(* CODESYS project Files.library
   Title: Files
   Version: 0.0.1
   Placeholder: Files
   Company: TomasRompotl

Project tree, tasks and I/O mapping:
  libraries: Events, * (TomasRompotl); MachineBase, * (TomasRompotl); Tc2_Standard, * (Beckhoff Automation GmbH); Tc2_System, * (Beckhoff Automation GmbH); Tc2_Utilities, * (Beckhoff Automation GmbH); Tc3_Module, * (Beckhoff Automation GmbH)
  File/
    function block Directory [ST]: Abort, Create, Cyclic, FileExists, FileNameList, CheckFileExists, List, Remove
    function block File [ST]: Busy, Cyclic, Done, Error, Read, Write
    function block FileRemover [ST]: Busy, Cyclic, Done, Error, Remove
  Version/
    global variables Global_Version
*)

// Version/Global_Version
{attribute 'TcGenerated'}
{attribute 'no-analysis'}
{attribute 'linkalways'}
// This function has been automatically generated from the project information.
VAR_GLOBAL CONSTANT
	{attribute 'const_non_replaced'}
	stLibVersion_Files : ST_LibVersion := (iMajor := 0, iMinor := 0, iBuild := 1, iRevision := 0, nFlags := 0, sVersion := '0.0.1');
END_VAR

// File/Directory
FUNCTION_BLOCK Directory
VAR
	creator : FB_CreateDir; // can only create on level of folder
	remover : FB_RemoveDir; // can only remove topmost folder. Not folder with folders.

	listDir : FB_EnumFindFileList;	
	listingFinishedTrigger : F_TRIG;
	fileListDone : BOOL;
	checkingFolder : BOOL;
	checkingFileExistence : BOOL;

	page : ARRAY[0..50 - 1] OF ST_FindFileEntry;
	_FileNameList : ARRAY[0..50 - 1] OF T_MaxString;
	_FileExists : BOOL;
	
	createDirectoryErrorTrig : R_TRIG;
	removeDirectoryErrorTrig : R_TRIG;
	listingDirectoryErrorTrig : R_TRIG;
	createDirectoryError : MessageEventLogger(TC_EVENTS.DirectoryEventClass.CreateDirectoryError);
	removeDirectoryError : MessageEventLogger(TC_EVENTS.DirectoryEventClass.RemoveDirectoryError);
	listingDirectoryError : MessageEventLogger(TC_EVENTS.DirectoryEventClass.ListDirectoryError);
END_VAR
VAR CONSTANT
	EntriesPerPage : INT := 50;
END_VAR

METHOD PRIVATE Abort
VAR_INPUT
END_VAR
listDir(
	bExecute := TRUE,
	eCmd := E_EnumCmdType.eEnumCmd_Abort
);
listDir(bExecute := FALSE);
END_METHOD

{attribute 'TcRpcEnable':='1'}
METHOD Create
VAR_INPUT
	path : T_MaxString;
END_VAR
creator(
	sPathName := path,
	bExecute := TRUE,
);
END_METHOD

METHOD Cyclic
VAR
	i : INT;
END_VAR
creator(bExecute := FALSE);
remover(bExecute := FALSE);

listDir(
	pFindList := ADR(page),
	cbFindList := SIZEOF(page)
);

listingFinishedTrigger(CLK := listDir.bBusy);
IF (listingFinishedTrigger.Q AND listDir.eCmd <> E_EnumCmdType.eEnumCmd_Abort) THEN

	listDir(bExecute := FALSE);
	fileListDone := TRUE;
	
	FOR i := 0 TO EntriesPerPage - 1 DO
		_FileNameList[i] := page[i].sFileName;
		
		IF (checkingFileExistence) THEN
			IF (page[i].fileAttributes.bDirectory = checkingFolder
				AND page[i].sFileName <> '') THEN
				_FileExists := TRUE;
			END_IF
		END_IF
	END_FOR
	
	IF (NOT listDir.bEOE) THEN
		Abort();
	END_IF
END_IF

createDirectoryErrorTrig(CLK := creator.bError);
removeDirectoryErrorTrig(CLK := remover.bError);
listingDirectoryErrorTrig(CLK := listDir.bError);
IF (createDirectoryErrorTrig.Q) THEN
	createDirectoryError.Arguments.Clear().AddStringByValue(creator.sPathName);
	createDirectoryError.Send();
END_IF
IF (removeDirectoryErrorTrig.Q) THEN
	removeDirectoryError.Arguments.Clear().AddStringByValue(remover.sPathName);
	removeDirectoryError.Send();
END_IF
IF (listingDirectoryErrorTrig.Q) THEN
	listingDirectoryError.Arguments.Clear().AddStringByValue(listDir.sPathName);
	listingDirectoryError.Send();
END_IF
END_METHOD

{attribute 'monitoring' := 'call'}
PROPERTY FileExists : BOOL
GET
FileExists := _FileExists;
END_GET
END_PROPERTY

{attribute 'monitoring' := 'call'}
PROPERTY FileNameList : REFERENCE TO ARRAY[0..49] OF T_MaxString
GET
FileNameList REF= _FileNameList;
END_GET
END_PROPERTY

METHOD CheckFileExists
VAR_INPUT
	path : T_MaxString;
	folder : BOOL; // FALSE = File, TRUE = Folder
END_VAR
IF (NOT listDir.bBusy) THEN
	
	List(path);
	
	_FileExists := FALSE;
	checkingFileExistence := TRUE;
	checkingFolder := folder;
END_IF
END_METHOD

 // Usage of * wildcard recommended
 // Add * to the end of path to list all files
METHOD List
VAR_INPUT
	path : T_MaxString;
END_VAR
IF (NOT listDir.bBusy) THEN
	
	checkingFileExistence := FALSE;
	fileListDone := FALSE;
	
	listDir(bExecute := FALSE);
	listDir(
		sPathName := path,
		eCmd := E_EnumCmdType.eEnumCmd_First,
		bExecute := TRUE
	);
END_IF
END_METHOD

METHOD Remove
VAR_INPUT
	path : T_MaxString;
END_VAR
remover(
	sPathName := path,
	bExecute := TRUE,
);
END_METHOD

END_FUNCTION_BLOCK

// File/File
FUNCTION_BLOCK File IMPLEMENTS Cyclic
VAR
	_Busy : BOOL;
	_Done : BOOL;
	_Error : BOOL;
	
	openRequest : BOOL;
	readRequest : BOOL;
	writeRequest : BOOL;
	appendMode : BOOL;
	filePath : T_MaxString;
	
	buffer : POINTER TO BYTE;
	bufferLength : UDINT;

	handle : UINT;
	opener : FB_FileOpen;
	closer : FB_FileClose;
	reader : FB_FileRead;
	writer : FB_FileWrite;
	
	fileState : (Waiting, OpenMode, Opening, Reading, Writing, Closing);
	openErrorTrigger : R_TRIG;
	readErrorTrigger : R_TRIG;
	writeErrorTrigger : R_TRIG;
	closeErrorTrigger : R_TRIG;
	
	notFoundError : MessageEventLogger(TC_EVENTS.FileEventClass.InvalidPath);
	fileOpenError : MessageEventLogger(TC_EVENTS.FileEventClass.OpenFileError);
	fileReadError : MessageEventLogger(TC_EVENTS.FileEventClass.ReadFileError);
	fileWriteError : MessageEventLogger(TC_EVENTS.FileEventClass.WriteFileError);
	fileCloseError : MessageEventLogger(TC_EVENTS.FileEventClass.CloseFileError);
END_VAR
VAR CONSTANT
	NotFoundErrorNumber : UDINT := 16#70C;
END_VAR

{attribute 'monitoring' := 'call'}
PROPERTY Busy : BOOL
GET
Busy := _Busy;
END_GET
END_PROPERTY

METHOD Cyclic
CASE fileState OF
	
	Waiting:
	
		IF (openRequest) THEN
			openRequest := FALSE;
			_Done := FALSE;
			
			fileState := OpenMode;
		END_IF
	
	OpenMode:
	
		IF (readRequest) THEN
			opener.nMode := FOPEN_MODEREAD;
		ELSIF (writeRequest) THEN
			IF (appendMode) THEN
				opener.nMode := FOPEN_MODEAPPEND;
			ELSE
				opener.nMode := FOPEN_MODEWRITE;
			END_IF
		END_IF
		
		opener.nMode := opener.nMode OR FOPEN_MODETEXT;

		fileState := Opening;
	
	Opening:
	
		opener(
			bExecute := NOT opener.bBusy,
			sPathName := filePath,
			hFile => handle,
		);
		
		IF (NOT opener.bExecute AND NOT opener.bBusy AND handle <> 0) THEN
			opener();
			IF (readRequest) THEN
				fileState := Reading;
			ELSIF (writeRequest) THEN
				fileState := Writing;
			END_IF
		END_IF
	
	Reading:
	
		reader(
			bExecute := NOT reader.bBusy,
			hFile := handle,
			pReadBuff := buffer,
			cbReadLen := bufferLength,
		);
		
		IF (NOT reader.bExecute AND NOT reader.bBusy) THEN
			fileState := Closing;
		END_IF
	
	Writing:
	
		writer(
			bExecute := NOT writer.bBusy,
			hFile := handle,
			pWriteBuff := buffer,
			cbWriteLen := bufferLength,
		);
		
		IF (NOT writer.bExecute AND NOT writer.bBusy) THEN
			fileState := Closing;
		END_IF
	
	Closing:
	
		IF (handle = 0) THEN
			fileState := Waiting;
		ELSE
			closer(
				bExecute := NOT closer.bBusy,
				hFile := handle,
			);
			
			IF (NOT closer.bExecute AND NOT closer.bBusy) THEN
				closer();
				handle := 0;
				_Done := TRUE;
				
				fileState := Waiting;
			END_IF
		END_IF
	
END_CASE

_Busy := fileState <> Waiting;

openErrorTrigger(CLK := opener.bError);
readErrorTrigger(CLK := reader.bError);
writeErrorTrigger(CLK := writer.bError);
closeErrorTrigger(CLK := closer.bError);
_Error := 
	openErrorTrigger.Q
	OR readErrorTrigger.Q
	OR writeErrorTrigger.Q
	OR closeErrorTrigger.Q
	;
IF (_Error) THEN
	openRequest := FALSE;
	readRequest := FALSE;
	writeRequest := FALSE;
	
	IF (openErrorTrigger.Q AND opener.nErrId = NotFoundErrorNumber) THEN
		notFoundError.Arguments.Clear().AddStringByValue(opener.sPathName);
		notFoundError.Send();
	ELSIF (openErrorTrigger.Q) THEN
		fileOpenError.Arguments.Clear().AddStringByValue(opener.sPathName);
		fileOpenError.Send();
	ELSIF (readErrorTrigger.Q) THEN
		fileReadError.Arguments.Clear().AddStringByValue(opener.sPathName);
		fileReadError.Send();
	ELSIF (openErrorTrigger.Q) THEN
		fileWriteError.Arguments.Clear().AddStringByValue(opener.sPathName);
		fileWriteError.Send();
	ELSIF (openErrorTrigger.Q) THEN
		fileCloseError.Arguments.Clear().AddStringByValue(opener.sPathName);
		fileCloseError.Send();
	END_IF
	
	IF (fileState > Waiting AND fileState < Closing) THEN
		fileState := Closing;
	END_IF
END_IF
END_METHOD

{attribute 'monitoring' := 'call'}
PROPERTY Done : BOOL
GET
Done := _Done;
END_GET
END_PROPERTY

{attribute 'monitoring' := 'call'}
PROPERTY Error : BOOL
GET
Error := _Error;
END_GET
END_PROPERTY

METHOD Read
VAR_INPUT
	buffer : POINTER TO BYTE;
	bufferLength : UDINT;
	filePath : T_MaxString;
END_VAR
IF (NOT _Busy) THEN
	THIS^.filePath := filePath;
	THIS^.buffer := buffer;
	THIS^.bufferLength := bufferLength;
	
	openRequest := TRUE;
	readRequest := TRUE;
	writeRequest := FALSE;
END_IF
END_METHOD

METHOD Write
VAR_INPUT
	buffer : POINTER TO BYTE;
	bufferLength : UDINT;
	filePath : T_MaxString;
	append : BOOL;
END_VAR
IF (NOT _Busy) THEN
	THIS^.filePath := filePath;
	THIS^.buffer := buffer;
	THIS^.bufferLength := bufferLength;
	
	openRequest := TRUE;
	writeRequest := TRUE;
	readRequest := FALSE;
	appendMode := append;
END_IF
END_METHOD

END_FUNCTION_BLOCK

// File/FileRemover
FUNCTION_BLOCK FileRemover IMPLEMENTS Cyclic
VAR
	remover : FB_FileDelete;
	
	removeErrorTrigger : R_TRIG;
	notFoundError : MessageEventLogger(TC_EVENTS.FileEventClass.InvalidPath);
	removeError : MessageEventLogger(TC_EVENTS.FileEventClass.RemoveFileError);
END_VAR
VAR CONSTANT
	NotFoundErrorNumber : UDINT := 16#70C;
END_VAR

{attribute 'monitoring' := 'call'}
PROPERTY Busy : BOOL
GET
Busy := remover.bBusy;
END_GET
END_PROPERTY

METHOD Cyclic
remover(bExecute := FALSE);

removeErrorTrigger(CLK := remover.bError);
IF (removeErrorTrigger.Q) THEN
	IF (remover.nErrId = NotFoundErrorNumber) THEN
		notFoundError.Arguments.Clear().AddStringByValue(remover.sPathName);
		notFoundError.Send();
	ELSE
		removeError.Arguments.Clear().AddStringByValue(remover.sPathName);
		removeError.Send();
	END_IF
END_IF
END_METHOD

{attribute 'monitoring' := 'call'}
PROPERTY Done : BOOL
GET
Done := NOT remover.bBusy;
END_GET
END_PROPERTY

{attribute 'monitoring' := 'call'}
PROPERTY Error : BOOL
GET
Error := remover.bError;
END_GET
END_PROPERTY

METHOD Remove
VAR_INPUT
	filePath : T_MaxString;
END_VAR
remover(
	sPathName := filePath,
	bExecute := TRUE
);
END_METHOD

END_FUNCTION_BLOCK
